// TIA Portal project "4 motor" (V16)

(* hardware
DEVICE "S7-1200 station_1"  S7-1200 Station
   slot 0: "Rack_0"  S7-1200 Rack  Rack  V1.0
   slot 1: "PLC_1"  CPU 1212C AC/DC/Rly  6ES7 212-1BE40-0XB0  V4.0
*)

// ===== PLC "PLC_1"  CPU 1212C AC/DC/Rly =====

VAR_GLOBAL   // PLC tag table "Default tag table"
   "stop" AT %I0.0 : Bool;
   "start" AT %I0.1 : Bool;
   "motor 1" AT %Q0.0 : Bool;
   "motor 2" AT %Q0.1 : Bool;
   "motor 3" AT %Q0.2 : Bool;
   "motor 4" AT %Q0.3 : Bool;
   "state 1" AT %M0.0 : Bool;
   "state 2" AT %M0.1 : Bool;
   "state 3" AT %M0.2 : Bool;
   "state 4" AT %M0.3 : Bool;
   "loop marker" AT %M0.4 : Bool;
END_VAR

// folder: System blocks/Program resources

DATA_BLOCK "T1"   // DB1
{ S7_Optimized_Access := 'TRUE' }
AUTHOR : Simatic
FAMILY : IEC
NAME : IEC_TMR
VERSION : 1.0
// stored: InstanceOfName IEC_TIMER
"IEC_TIMER"
BEGIN
END_DATA_BLOCK

DATA_BLOCK "T2"   // DB2
{ S7_Optimized_Access := 'TRUE' }
AUTHOR : Simatic
FAMILY : IEC
NAME : IEC_TMR
VERSION : 1.0
// stored: InstanceOfName IEC_TIMER
"IEC_TIMER"
BEGIN
END_DATA_BLOCK

DATA_BLOCK "T3"   // DB3
{ S7_Optimized_Access := 'TRUE' }
AUTHOR : Simatic
FAMILY : IEC
NAME : IEC_TMR
VERSION : 1.0
// stored: InstanceOfName IEC_TIMER
"IEC_TIMER"
BEGIN
END_DATA_BLOCK

DATA_BLOCK "T4"   // DB4
{ S7_Optimized_Access := 'TRUE' }
AUTHOR : Simatic
FAMILY : IEC
NAME : IEC_TMR
VERSION : 1.0
// stored: InstanceOfName IEC_TIMER
"IEC_TIMER"
BEGIN
END_DATA_BLOCK

// folder: (top level)

ORGANIZATION_BLOCK "Main"   // OB1, LAD, ProgramCycle
TITLE = "Main Program Sweep (Cycle)"
{ S7_Optimized_Access := 'TRUE' }
VERSION : 0.1
   VAR_INPUT
      Initial_Call : Bool;   // Initial call of this OB
      Remanence : Bool;   // =True, if remanent data are available
   END_VAR
BEGIN

REGION Network 1
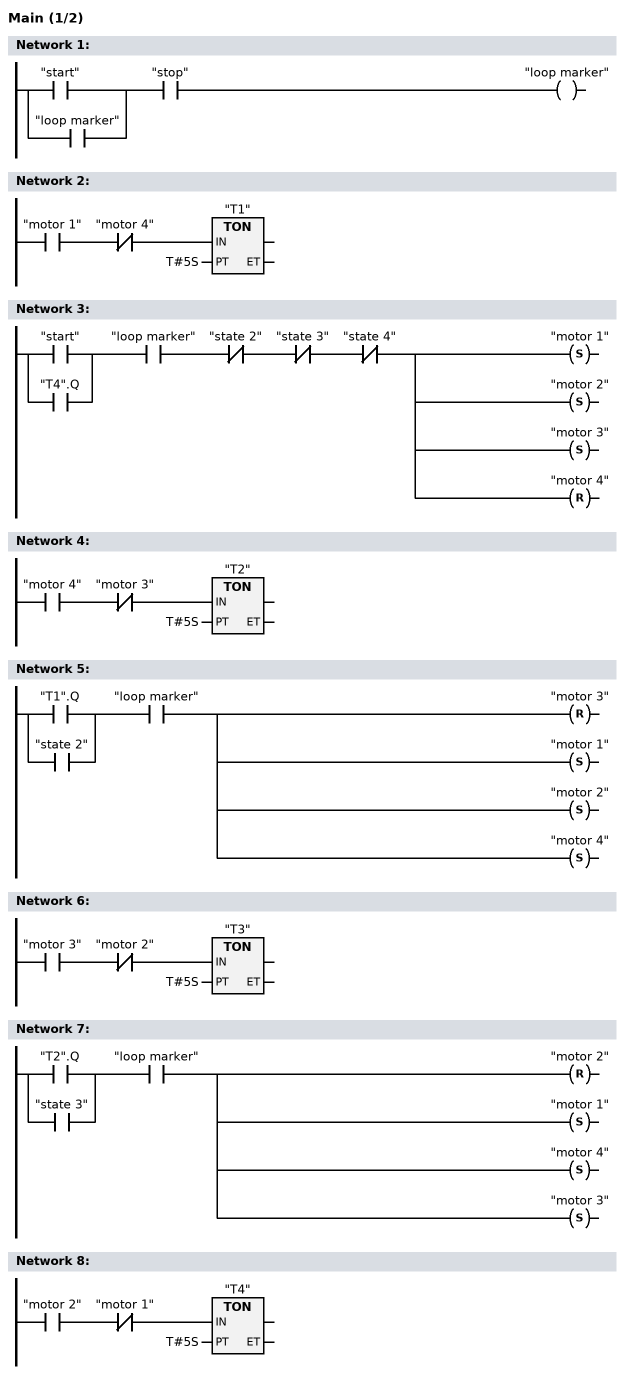
   RUNG wire#powerrail
      Contact( "start" )
      wire#w1
      Contact( "stop" )
      Coil( "loop marker" )
   END_RUNG
   RUNG wire#powerrail
      Contact( "loop marker" )
   END_RUNG wire#w1
   // the same network as SCL:
   "loop marker" := ("start" OR "loop marker") AND "stop";
END_REGION

REGION Network 2
   "T1".TON(IN := "motor 1" AND NOT "motor 4", PT := T#5S);
END_REGION

REGION Network 3
   RUNG wire#powerrail
      Contact( "start" )
      wire#w1
      Contact( "loop marker" )
      I_Contact( "state 2" )
      I_Contact( "state 3" )
      I_Contact( "state 4" )
      wire#w2
      S_Coil( "motor 1" )
   END_RUNG
   RUNG wire#powerrail
      Contact( "T4".Q )
   END_RUNG wire#w1
   RUNG wire#w2
      S_Coil( "motor 2" )
   END_RUNG
   RUNG wire#w2
      S_Coil( "motor 3" )
   END_RUNG
   RUNG wire#w2
      R_Coil( "motor 4" )
   END_RUNG
   // the same network as SCL:
   IF ("start" OR "T4".Q) AND "loop marker" AND NOT "state 2" AND NOT "state 3" AND NOT "state 4" THEN
       "motor 1" := TRUE;
       "motor 2" := TRUE;
       "motor 3" := TRUE;
       "motor 4" := FALSE;
   END_IF;
END_REGION

REGION Network 4
   "T2".TON(IN := "motor 4" AND NOT "motor 3", PT := T#5S);
END_REGION

REGION Network 5
   RUNG wire#powerrail
      Contact( "T1".Q )
      wire#w1
      Contact( "loop marker" )
      wire#w2
      R_Coil( "motor 3" )
   END_RUNG
   RUNG wire#powerrail
      Contact( "state 2" )
   END_RUNG wire#w1
   RUNG wire#w2
      S_Coil( "motor 1" )
   END_RUNG
   RUNG wire#w2
      S_Coil( "motor 2" )
   END_RUNG
   RUNG wire#w2
      S_Coil( "motor 4" )
   END_RUNG
   // the same network as SCL:
   IF ("T1".Q OR "state 2") AND "loop marker" THEN
       "motor 3" := FALSE;
       "motor 1" := TRUE;
       "motor 2" := TRUE;
       "motor 4" := TRUE;
   END_IF;
END_REGION

REGION Network 6
   "T3".TON(IN := "motor 3" AND NOT "motor 2", PT := T#5S);
END_REGION

REGION Network 7
   RUNG wire#powerrail
      Contact( "T2".Q )
      wire#w1
      Contact( "loop marker" )
      wire#w2
      R_Coil( "motor 2" )
   END_RUNG
   RUNG wire#powerrail
      Contact( "state 3" )
   END_RUNG wire#w1
   RUNG wire#w2
      S_Coil( "motor 1" )
   END_RUNG
   RUNG wire#w2
      S_Coil( "motor 4" )
   END_RUNG
   RUNG wire#w2
      S_Coil( "motor 3" )
   END_RUNG
   // the same network as SCL:
   IF ("T2".Q OR "state 3") AND "loop marker" THEN
       "motor 2" := FALSE;
       "motor 1" := TRUE;
       "motor 4" := TRUE;
       "motor 3" := TRUE;
   END_IF;
END_REGION

REGION Network 8
   "T4".TON(IN := "motor 2" AND NOT "motor 1", PT := T#5S);
END_REGION

REGION Network 9
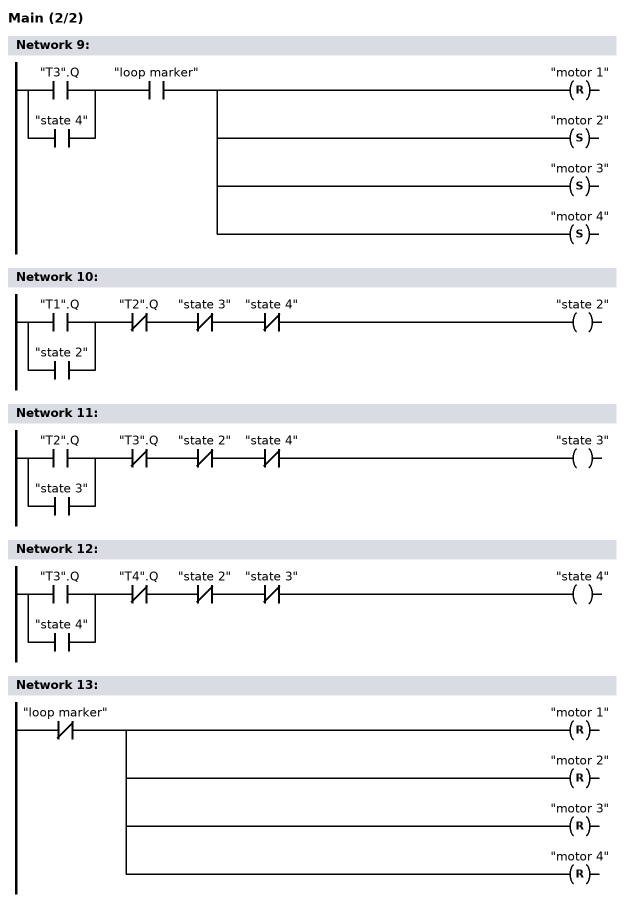
   RUNG wire#powerrail
      Contact( "T3".Q )
      wire#w1
      Contact( "loop marker" )
      wire#w2
      R_Coil( "motor 1" )
   END_RUNG
   RUNG wire#powerrail
      Contact( "state 4" )
   END_RUNG wire#w1
   RUNG wire#w2
      S_Coil( "motor 2" )
   END_RUNG
   RUNG wire#w2
      S_Coil( "motor 3" )
   END_RUNG
   RUNG wire#w2
      S_Coil( "motor 4" )
   END_RUNG
   // the same network as SCL:
   IF ("T3".Q OR "state 4") AND "loop marker" THEN
       "motor 1" := FALSE;
       "motor 2" := TRUE;
       "motor 3" := TRUE;
       "motor 4" := TRUE;
   END_IF;
END_REGION

REGION Network 10
   RUNG wire#powerrail
      Contact( "T1".Q )
      wire#w1
      I_Contact( "T2".Q )
      I_Contact( "state 3" )
      I_Contact( "state 4" )
      Coil( "state 2" )
   END_RUNG
   RUNG wire#powerrail
      Contact( "state 2" )
   END_RUNG wire#w1
   // the same network as SCL:
   "state 2" := ("T1".Q OR "state 2") AND NOT "T2".Q AND NOT "state 3" AND NOT "state 4";
END_REGION

REGION Network 11
   RUNG wire#powerrail
      Contact( "T2".Q )
      wire#w1
      I_Contact( "T3".Q )
      I_Contact( "state 2" )
      I_Contact( "state 4" )
      Coil( "state 3" )
   END_RUNG
   RUNG wire#powerrail
      Contact( "state 3" )
   END_RUNG wire#w1
   // the same network as SCL:
   "state 3" := ("T2".Q OR "state 3") AND NOT "T3".Q AND NOT "state 2" AND NOT "state 4";
END_REGION

REGION Network 12
   RUNG wire#powerrail
      Contact( "T3".Q )
      wire#w1
      I_Contact( "T4".Q )
      I_Contact( "state 2" )
      I_Contact( "state 3" )
      Coil( "state 4" )
   END_RUNG
   RUNG wire#powerrail
      Contact( "state 4" )
   END_RUNG wire#w1
   // the same network as SCL:
   "state 4" := ("T3".Q OR "state 4") AND NOT "T4".Q AND NOT "state 2" AND NOT "state 3";
END_REGION

REGION Network 13
   RUNG wire#powerrail
      I_Contact( "loop marker" )
      wire#w1
      R_Coil( "motor 1" )
   END_RUNG
   RUNG wire#w1
      R_Coil( "motor 2" )
   END_RUNG
   RUNG wire#w1
      R_Coil( "motor 3" )
   END_RUNG
   RUNG wire#w1
      R_Coil( "motor 4" )
   END_RUNG
   // the same network as SCL:
   IF NOT "loop marker" THEN
       "motor 1" := FALSE;
       "motor 2" := FALSE;
       "motor 3" := FALSE;
       "motor 4" := FALSE;
   END_IF;
END_REGION
END_ORGANIZATION_BLOCK